// Mitsubishi GX Works2 project: theory2   PLC: FX3G

// global labels: Global1
VAR_GLOBAL
  startDay AT X007 : BOOL;
  Y_7 AT Y007 : BOOL;
END_VAR
VAR_GLOBAL CONSTANT
  startingFule : INT := 400;
END_VAR
VAR_GLOBAL
  currentFule AT D1100 : INT;
END_VAR
VAR_GLOBAL CONSTANT
  con_300 : INT := 300;
END_VAR
VAR_GLOBAL
  notEnoughFule AT M0 : BOOL;
  stopDay AT Y000 : BOOL;
  fullOfApples AT CC1 : BOOL;
END_VAR
VAR_GLOBAL CONSTANT
  boxes : INT := 5;
END_VAR
VAR_GLOBAL
  fulll AT CS1 : BOOL;
  endOfDay AT M2 : BOOL;
  anotherBoxOfAppels AT X000 : BOOL;
  TC2 AT TC2 : BOOL;
  tc_2 AT TC2 : BOOL;
END_VAR
VAR_GLOBAL CONSTANT
  con600 : WORD;
  con390 : WORD;
END_VAR
VAR_GLOBAL
  filledFule AT M4 : BOOL;
END_VAR
VAR_GLOBAL CONSTANT
  con_10 : INT := 10;
END_VAR
VAR_GLOBAL
  ts_2 AT TS2 : BOOL;
END_VAR
VAR_GLOBAL CONSTANT
  con4 : INT := 40;
END_VAR
VAR_GLOBAL
  putInFule AT X004 : BOOL;
END_VAR

// task Task_01 (event TRUE, interval 0, priority 31): POU_01

PROGRAM POU_01
(* structured ladder/FBD written out as ST: instructions are called as NAME(EN, inputs, outputs); _pN, _eN, _tN stand for wires *)
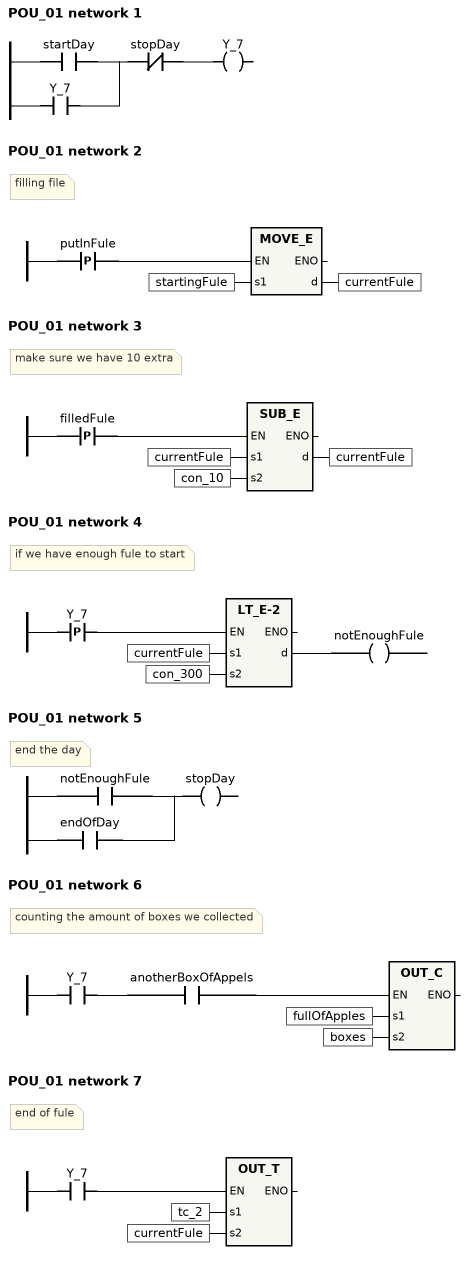
(* network 1 *)
Y_7 := (startDay OR Y_7) AND NOT stopDay;
(* network 2 *)
(* filling file *)
MOVE_E(LDP(TRUE, putInFule), startingFule, currentFule);
(* network 3 *)
(* make sure we have 10 extra *)
SUB_E(LDP(TRUE, filledFule), currentFule, con_10, currentFule);
(* network 4 *)
(* if we have enough fule to start *)
LT_E(LDP(TRUE, Y_7), currentFule, con_300, _t1);
notEnoughFule := _t1;
(* network 5 *)
(* end the day *)
stopDay := notEnoughFule OR endOfDay;
(* network 6 *)
(* counting the amount of boxes we collected *)
OUT_C(Y_7 AND anotherBoxOfAppels, fullOfApples, boxes);
(* network 7 *)
(* end of fule *)
OUT_T(Y_7, tc_2, currentFule);
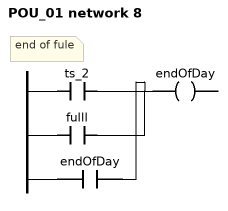
(* network 8 *)
(* end of fule *)
endOfDay := ts_2 OR fulll OR endOfDay;
END_PROGRAM
